// Registered entity handle.
INTERFACE I_Entity EXTENDS _I_Entity

// Raw discoverable interface for __QUERYINTERFACE.
PROPERTY Raw : I_Generic
GET
END_GET
END_PROPERTY

END_INTERFACE

(* stored: Version 1.1.0.1
   Itf I_Entity: Id {34f52675-879c-44cb-b9cd-6851c154fd0c}
   Property Raw: Id {304f904b-75c2-47dc-94c7-d14b30af4057}
   Get Get: Id {65bf2b6b-3eaa-44ba-8b9d-310345aa0739} *)
